// TwinCAT 3 PLC project SimulateAxisLag
// ProgramVersion: 3.1.4024.0
// libraries:
//   Tc2_MC2, * (Beckhoff Automation GmbH)
//   Tc2_Standard, * (Beckhoff Automation GmbH)
//   Tc2_System, * (Beckhoff Automation GmbH)
//   Tc3_Module, * (Beckhoff Automation GmbH)
// project tree:
//   / PlcTask.TcTTO
//   POUs/ MAIN.TcPOU
// real-time tasks:
//   TASK PlcTask: cycle T#1ms, priority 20, ADS port 350
// motion (NC):
//   TASK NC-Task 1 SAF: cycle T#2ms, priority 4, ADS port 501
//   TASK NC-Task 1 SVB: cycle T#10ms, priority 8, ADS port 511
//   AXIS Axis 1 (id 1)
//     OtherSettings: ErrorReactionMode=1, ErrorReactionDelay=0.03, AllowMotionCmdToSlave=true
//     encoder EncType=4
//       EncPara: ScaleFactorNumerator=0.01, MaxCount=#x0000ffff
//         ActPosCorrection: Enable=true
//         Inc: RefMode=2
//         TimeComp: TimeCompMode=1, AdditionalTimeShift=55000
//     drive DrvType=13
//       Analog: VeloReferenz=2000, TorqueSetpointScale=10, ScaleFactorActTorque=0.1
//       TimeComp: TimeCompMode=1, DriveDelayCycles=3, TaskDelayCycles=1
//     controller CtrType=1
//       CtrPara: PriorControlFactor=1
//         PosDiffControl: Range=100, Time=0.1
//         Observer: BandWidth=20
// variable links:
//   SimulateAxisLag Instance <-> NC-Task 1 SAF/Axes/Axis 1
//     PlcTask Inputs/MAIN.ax.NcToPlc <-> Outputs/ToPlc
//     PlcTask Outputs/MAIN.q_ui1 <-> Enc/Inputs/In/nDataIn1[0]
//     PlcTask Outputs/MAIN.q_ui2 <-> Enc/Inputs/In/nDataIn1[1]

CONFIGURATION SimulateAxisLag
    RESOURCE PLC ON TwinCAT3
        TASK PlcTask(INTERVAL := T#1ms, PRIORITY := 20);
        PROGRAM MAIN WITH PlcTask : MAIN;
    END_RESOURCE
END_CONFIGURATION

// ---- POUs/MAIN.TcPOU
PROGRAM MAIN
VAR
	q_ui1, q_ui2 AT%Q*: UINT;
	noLag: BOOL := TRUE;;
	noSim: BOOL := TRUE;;
	ax: axis_ref;
	actPos : LREAL;
	actPosIn : LREAL;
END_VAR

(*
===========================DISCLAIMER=============================
All sample code provided by Beckhoff Automation LLC are
 for illustrative purposes only and are provided “as is”
 and without any warranties, express or implied. Actual
 implementations in applications will vary significantly.
 Beckhoff Automation LLC shall have no liability for, and
 does not waive any rights in relation to, any code samples
 that it provides or the use of such code samples for any purpose.
*)

ax.ReadStatus();
IF noLag THEN // set to false to cause lag on when jogging the axis
	q_ui1 := TO_UINT(TO_DINT(ax.NcToPlc.SetPos / 0.01) MOD 65535);
	q_ui2 := TO_UINT(TO_DINT(ax.NcToPlc.SetPos / 0.01) -  q_ui1);	
ELSIF noSim THEN
	q_ui1 := TO_UINT(TO_DINT(actPosIn / 0.01) MOD 65535);
	q_ui2 := TO_UINT(TO_DINT(actPosIn / 0.01) -  q_ui1);	
ELSE
	q_ui1 := TO_UINT(TO_DINT(actPos / 0.01) MOD 65535);
	q_ui2 := TO_UINT(TO_DINT(actPos / 0.01) -  q_ui1);
END_IF

END_PROGRAM
